SYSTEM Boiler
  (* Version 1.0, Author, 4DIAC-Consortium *)
  APPLICATION MyBoiler
    FBS
      IN_ANY_1 : IN_ANY(QI := 1, TYPE := LREAL, IVAL := 0);
      OUT_ANY : OUT_ANY(QI := 1, TYPE := LREAL, IVAL := 0);
      LREAL2LREAL_0 : LREAL2LREAL;
      FB_LABEL_0 : FB_LABEL(QI := 1, LABEL := Steam Removal (0..10));
      LREAL2LREAL_2 : LREAL2LREAL;
      OUT_ANY_0 : OUT_ANY(QI := 1, TYPE := LREAL, IVAL := 1);
      FB_LABEL_1 : FB_LABEL(QI := 1, LABEL := Actual Fill Level);
      FB_LABEL_2 : FB_LABEL(QI := 1, LABEL := Actual Feed Water Flow);
      OUT_ANY_1 : OUT_ANY(QI := 1, TYPE := LREAL, IVAL := 1);
      FB_LABEL_3 : FB_LABEL(QI := 1, LABEL := Actual Steam Flow);
      LREAL2LREAL_5 : LREAL2LREAL;
      IN_ANY : IN_ANY(QI := 1, TYPE := LREAL, IVAL := 0);
      FB_LABEL : FB_LABEL(QI := 1, LABEL := Set Fill Level (0..1000));
      LREAL2LREAL : LREAL2LREAL;
      LREAL2LREAL_1 : LREAL2LREAL;
      FlowController : FlowController;
      ControlComputation : ControlComputation;
      BasicAO : BasicAO(minEng := 0, maxEng := 10, minRaw := 0, maxRaw := 16#FFFF);
      FeedWaterValve : QW(QI := 1, PARAMS := %watervalve%);
      SteamValve : QW(QI := 1, PARAMS := %steamvalve%);
      BasicAO_0 : BasicAO(minEng := 0, maxEng := 10, minRaw := 0, maxRaw := 16#FFFF);
      LC : BasicPID(bReset := 0, fCtrlCycleTime := 0.01, fTv := 0, fTd := 0.01, fKp := 1, fTn := 0);
      BasicAI_1 : BasicAI(minEng := 0, maxEng := 1000, minRaw := 0, maxRaw := 16#FFFF);
      TankLevel : IW(QI := 1, PARAMS := %tanklevel%);
      E_CYCLE : E_CYCLE(DT := T#100ms);
      BasicAI_2 : BasicAI(minEng := 0, maxEng := 10, minRaw := 0, maxRaw := 16#FFFF);
      SteamFlow : IW(QI := 1, PARAMS := %steamflow%);
      IW : IW(QI := 1, PARAMS := %feedwaterflow%);
      BasicAI_3 : BasicAI(minEng := 0, maxEng := 10, minRaw := 0, maxRaw := 16#FFFF);
      LREAL2LREAL_3 : LREAL2LREAL;
      OUT_ANY_2 : OUT_ANY(QI := 1, TYPE := LREAL, IVAL := 0);
      FB_LABEL_4 : FB_LABEL(QI := 1, LABEL := Feed Water Valve);
      IN_ANY_0 : IN_ANY(TYPE := LREAL, IVAL := 0);
    END_FBS
    EVENT_CONNECTIONS
      LREAL2LREAL_0.CNF TO OUT_ANY.REQ;
      FB_LABEL_0.INITO TO IN_ANY_1.INIT;
      OUT_ANY.CNF TO LREAL2LREAL_2.REQ;
      LREAL2LREAL_2.CNF TO OUT_ANY_0.REQ;
      FB_LABEL_1.INITO TO OUT_ANY.INIT;
      OUT_ANY.INITO TO FB_LABEL_2.INIT;
      FB_LABEL_2.INITO TO OUT_ANY_0.INIT;
      FB_LABEL_3.INITO TO OUT_ANY_1.INIT;
      OUT_ANY_0.INITO TO FB_LABEL_3.INIT;
      LREAL2LREAL_5.CNF TO OUT_ANY_1.REQ;
      OUT_ANY_0.CNF TO LREAL2LREAL_5.REQ;
      FB_LABEL.INITO TO IN_ANY.INIT;
      IN_ANY.INITO TO FB_LABEL_0.INIT;
      IN_ANY.IND TO LREAL2LREAL.REQ;
      LREAL2LREAL.CNF TO IN_ANY_1.REQ;
      IN_ANY_1.IND TO LREAL2LREAL_1.REQ;
      ControlComputation.CNF TO FlowController.REQ;
      FlowController.CNF TO BasicAO.REQ;
      BasicAO.CNF TO FeedWaterValve.REQ;
      BasicAO.INITO TO FeedWaterValve.INIT;
      BasicAO_0.CNF TO SteamValve.REQ;
      BasicAO_0.INITO TO SteamValve.INIT;
      LREAL2LREAL_1.CNF TO BasicAO_0.REQ;
      TankLevel.INITO TO BasicAI_1.INIT;
      TankLevel.CNF TO BasicAI_1.REQ;
      E_CYCLE.EO TO TankLevel.REQ;
      LC.CNF TO ControlComputation.REQ;
      SteamFlow.CNF TO BasicAI_2.REQ;
      IW.CNF TO BasicAI_3.REQ;
      BasicAI_1.CNF TO IW.REQ;
      BasicAI_2.CNF TO LC.REQ;
      OUT_ANY_1.CNF TO LREAL2LREAL_3.REQ;
      LREAL2LREAL_3.CNF TO OUT_ANY_2.REQ;
      OUT_ANY_1.INITO TO FB_LABEL_4.INIT;
      FB_LABEL_4.INITO TO OUT_ANY_2.INIT;
      IW.INITO TO BasicAI_3.INIT;
      SteamFlow.INITO TO BasicAI_2.INIT;
      SteamValve.INITO TO BasicAO.INIT;
      BasicAI_3.CNF TO SteamFlow.REQ;
      BasicAI_3.INITO TO SteamFlow.INIT;
      BasicAI_1.INITO TO IW.INIT;
      BasicAI_2.INITO TO BasicAO_0.INIT;
      FeedWaterValve.INITO TO E_CYCLE.START;
    END_CONNECTIONS
    DATA_CONNECTIONS
      LREAL2LREAL_0.OUT TO OUT_ANY.IN;
      LREAL2LREAL_2.OUT TO OUT_ANY_0.IN;
      LREAL2LREAL_5.OUT TO OUT_ANY_1.IN;
      FB_LABEL_0.QO TO IN_ANY_1.QI;
      FB_LABEL.QO TO IN_ANY.QI;
      IN_ANY.OUT TO LREAL2LREAL.IN;
      IN_ANY_1.OUT TO LREAL2LREAL_1.IN;
      ControlComputation.ControlOut TO FlowController.Setpoint;
      BasicAO.Out TO FeedWaterValve.OUT;
      FlowController.ControlOut TO BasicAO.Val;
      BasicAO_0.Out TO SteamValve.OUT;
      LREAL2LREAL_1.OUT TO BasicAO_0.Val;
      LREAL2LREAL.OUT TO LC.fSetpointValue;
      TankLevel.IN TO BasicAI_1.Val;
      LC.fCtrlOutput TO ControlComputation.Input1;
      BasicAI_1.Out TO LC.fActualValue;
      SteamFlow.IN TO BasicAI_2.Val;
      IW.IN TO BasicAI_3.Val;
      BasicAI_2.Out TO ControlComputation.Input3;
      BasicAI_3.Out TO ControlComputation.Input2;
      LREAL2LREAL_3.OUT TO OUT_ANY_2.IN;
      FlowController.ControlOut TO LREAL2LREAL_3.IN;
      BasicAI_2.Out TO LREAL2LREAL_5.IN;
      BasicAI_1.Out TO LREAL2LREAL_0.IN;
      BasicAI_3.Out TO LREAL2LREAL_2.IN;
    END_CONNECTIONS
  END_APPLICATION
  APPLICATION globals
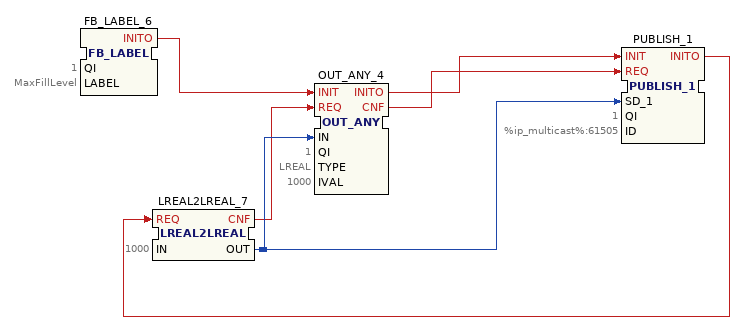
    FBS
      LREAL2LREAL_7 : LREAL2LREAL(IN := 1000);
      FB_LABEL_6 : FB_LABEL(QI := 1, LABEL := MaxFillLevel);
      OUT_ANY_4 : OUT_ANY(QI := 1, TYPE := LREAL, IVAL := 1000);
      PUBLISH_1 : PUBLISH_1(QI := 1, ID := %ip_multicast%:61505);
    END_FBS
    EVENT_CONNECTIONS
      OUT_ANY_4.INITO TO PUBLISH_1.INIT;
      FB_LABEL_6.INITO TO OUT_ANY_4.INIT;
      PUBLISH_1.INITO TO LREAL2LREAL_7.REQ;
      LREAL2LREAL_7.CNF TO OUT_ANY_4.REQ;
      OUT_ANY_4.CNF TO PUBLISH_1.REQ;
    END_CONNECTIONS
    DATA_CONNECTIONS
      LREAL2LREAL_7.OUT TO OUT_ANY_4.IN;
      LREAL2LREAL_7.OUT TO PUBLISH_1.SD_1;
    END_CONNECTIONS
  END_APPLICATION
  APPLICATION BoilerModel
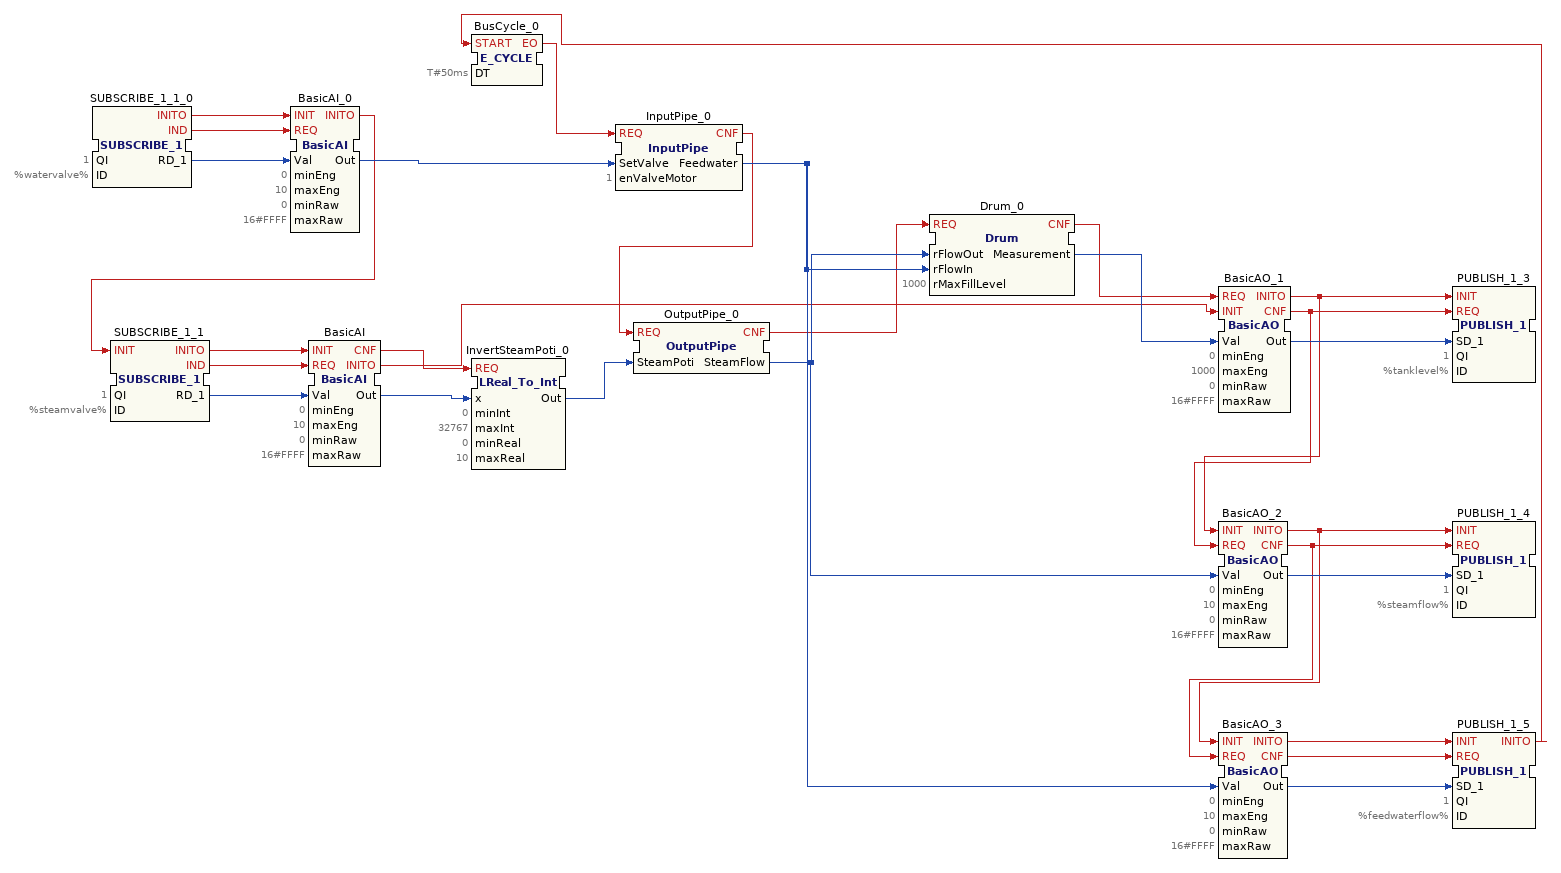
    FBS
      OutputPipe_0 : OutputPipe;
      Drum_0 : Drum(rMaxFillLevel := 1000);
      BusCycle_0 : E_CYCLE(DT := T#50ms);
      InvertSteamPoti_0 : LReal_To_Int(minInt := 0, maxInt := 32767, minReal := 0, maxReal := 10);
      InputPipe_0 : InputPipe(enValveMotor := 1);
      SUBSCRIBE_1_1 : SUBSCRIBE_1(QI := 1, ID := %steamvalve%);
      BasicAI : BasicAI(minEng := 0, maxEng := 10, minRaw := 0, maxRaw := 16#FFFF);
      SUBSCRIBE_1_1_0 : SUBSCRIBE_1(QI := 1, ID := %watervalve%);
      BasicAI_0 : BasicAI(minEng := 0, maxEng := 10, minRaw := 0, maxRaw := 16#FFFF);
      BasicAO_1 : BasicAO(minEng := 0, maxEng := 1000, minRaw := 0, maxRaw := 16#FFFF);
      BasicAO_2 : BasicAO(minEng := 0, maxEng := 10, minRaw := 0, maxRaw := 16#FFFF);
      BasicAO_3 : BasicAO(minEng := 0, maxEng := 10, minRaw := 0, maxRaw := 16#FFFF);
      PUBLISH_1_3 : PUBLISH_1(QI := 1, ID := %tanklevel%);
      PUBLISH_1_4 : PUBLISH_1(QI := 1, ID := %steamflow%);
      PUBLISH_1_5 : PUBLISH_1(QI := 1, ID := %feedwaterflow%);
    END_FBS
    EVENT_CONNECTIONS
      SUBSCRIBE_1_1.INITO TO BasicAI.INIT;
      SUBSCRIBE_1_1.IND TO BasicAI.REQ;
      SUBSCRIBE_1_1_0.INITO TO BasicAI_0.INIT;
      SUBSCRIBE_1_1_0.IND TO BasicAI_0.REQ;
      BasicAI.CNF TO InvertSteamPoti_0.REQ;
      BasicAO_1.INITO TO BasicAO_2.INIT;
      BasicAO_2.INITO TO BasicAO_3.INIT;
      BasicAO_1.CNF TO BasicAO_2.REQ;
      BasicAO_2.CNF TO BasicAO_3.REQ;
      BasicAO_1.INITO TO PUBLISH_1_3.INIT;
      BasicAO_1.CNF TO PUBLISH_1_3.REQ;
      BasicAO_2.INITO TO PUBLISH_1_4.INIT;
      BasicAO_2.CNF TO PUBLISH_1_4.REQ;
      BasicAO_3.INITO TO PUBLISH_1_5.INIT;
      BasicAO_3.CNF TO PUBLISH_1_5.REQ;
      BusCycle_0.EO TO InputPipe_0.REQ;
      OutputPipe_0.CNF TO Drum_0.REQ;
      InputPipe_0.CNF TO OutputPipe_0.REQ;
      BasicAI_0.INITO TO SUBSCRIBE_1_1.INIT;
      Drum_0.CNF TO BasicAO_1.REQ;
      PUBLISH_1_5.INITO TO BusCycle_0.START;
      BasicAI.INITO TO BasicAO_1.INIT;
    END_CONNECTIONS
    DATA_CONNECTIONS
      OutputPipe_0.SteamFlow TO Drum_0.rFlowOut;
      InputPipe_0.Feedwater TO Drum_0.rFlowIn;
      InvertSteamPoti_0.Out TO OutputPipe_0.SteamPoti;
      SUBSCRIBE_1_1.RD_1 TO BasicAI.Val;
      SUBSCRIBE_1_1_0.RD_1 TO BasicAI_0.Val;
      BasicAI_0.Out TO InputPipe_0.SetValve;
      BasicAI.Out TO InvertSteamPoti_0.x;
      BasicAO_1.Out TO PUBLISH_1_3.SD_1;
      BasicAO_2.Out TO PUBLISH_1_4.SD_1;
      BasicAO_3.Out TO PUBLISH_1_5.SD_1;
      Drum_0.Measurement TO BasicAO_1.Val;
      InputPipe_0.Feedwater TO BasicAO_3.Val;
      OutputPipe_0.SteamFlow TO BasicAO_2.Val;
    END_CONNECTIONS
  END_APPLICATION
  DEVICE HMI : FBRT_WINDOW(BOUNDS := [200,200,268,500], GRID := [3,1], MGR_ID := "localhost:61505")
    {SET_ATTRIBUTE(Profile, HOLOBLOC)}
    RESOURCE VIS_IN : PANEL_RESOURCE
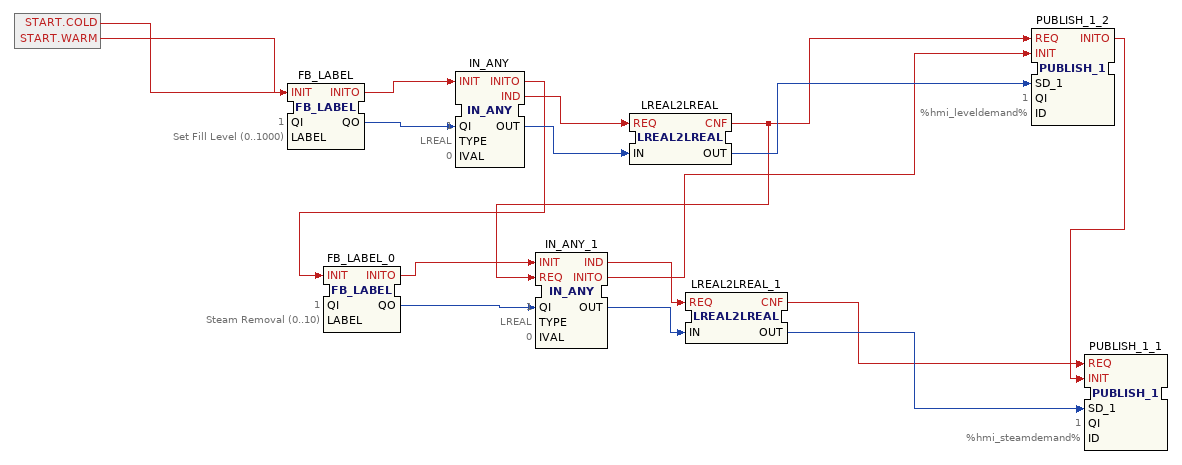
      FBS
        IN_ANY_1 : IN_ANY(QI := 1, TYPE := LREAL, IVAL := 0);
        FB_LABEL_0 : FB_LABEL(QI := 1, LABEL := Steam Removal (0..10));
        IN_ANY : IN_ANY(QI := 1, TYPE := LREAL, IVAL := 0);
        FB_LABEL : FB_LABEL(QI := 1, LABEL := Set Fill Level (0..1000));
        LREAL2LREAL : LREAL2LREAL;
        LREAL2LREAL_1 : LREAL2LREAL;
        PUBLISH_1_1 : PUBLISH_1(QI := 1, ID := %hmi_steamdemand%);
        PUBLISH_1_2 : PUBLISH_1(QI := 1, ID := %hmi_leveldemand%);
      END_FBS
      EVENT_CONNECTIONS
        FB_LABEL_0.INITO TO IN_ANY_1.INIT;
        IN_ANY.INITO TO FB_LABEL_0.INIT;
        FB_LABEL.INITO TO IN_ANY.INIT;
        IN_ANY.IND TO LREAL2LREAL.REQ;
        LREAL2LREAL.CNF TO IN_ANY_1.REQ;
        START.COLD TO FB_LABEL.INIT;
        START.WARM TO FB_LABEL.INIT;
        IN_ANY_1.IND TO LREAL2LREAL_1.REQ;
        LREAL2LREAL_1.CNF TO PUBLISH_1_1.REQ;
        LREAL2LREAL.CNF TO PUBLISH_1_2.REQ;
        IN_ANY_1.INITO TO PUBLISH_1_2.INIT;
        PUBLISH_1_2.INITO TO PUBLISH_1_1.INIT;
      END_CONNECTIONS
      DATA_CONNECTIONS
        FB_LABEL_0.QO TO IN_ANY_1.QI;
        FB_LABEL.QO TO IN_ANY.QI;
        IN_ANY.OUT TO LREAL2LREAL.IN;
        IN_ANY_1.OUT TO LREAL2LREAL_1.IN;
        LREAL2LREAL_1.OUT TO PUBLISH_1_1.SD_1;
        LREAL2LREAL.OUT TO PUBLISH_1_2.SD_1;
      END_CONNECTIONS
    END_RESOURCE
    RESOURCE VIS_OUT : PANEL_RESOURCE
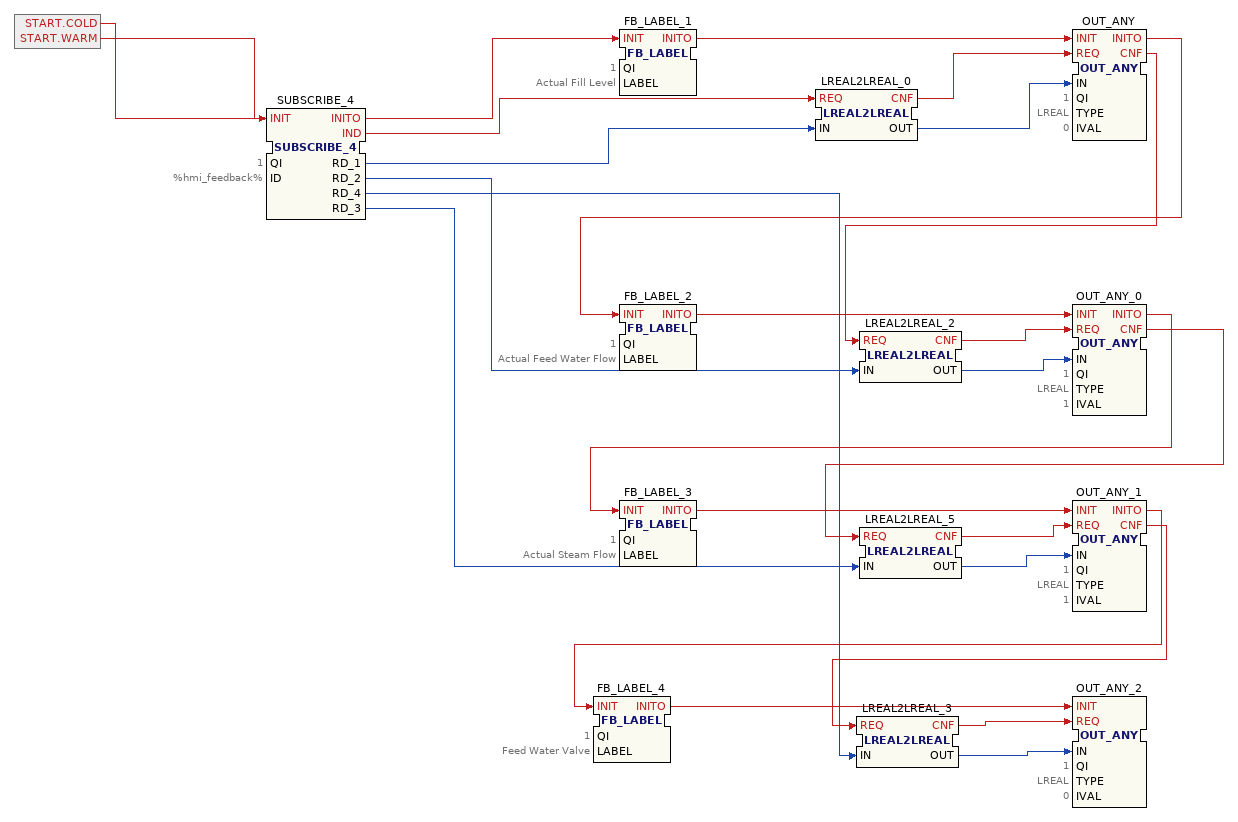
      FBS
        SUBSCRIBE_4 : SUBSCRIBE_4(QI := 1, ID := %hmi_feedback%);
        FB_LABEL_1 : FB_LABEL(QI := 1, LABEL := Actual Fill Level);
        LREAL2LREAL_0 : LREAL2LREAL;
        OUT_ANY : OUT_ANY(QI := 1, TYPE := LREAL, IVAL := 0);
        FB_LABEL_2 : FB_LABEL(QI := 1, LABEL := Actual Feed Water Flow);
        LREAL2LREAL_2 : LREAL2LREAL;
        OUT_ANY_0 : OUT_ANY(QI := 1, TYPE := LREAL, IVAL := 1);
        FB_LABEL_3 : FB_LABEL(QI := 1, LABEL := Actual Steam Flow);
        LREAL2LREAL_5 : LREAL2LREAL;
        OUT_ANY_1 : OUT_ANY(QI := 1, TYPE := LREAL, IVAL := 1);
        FB_LABEL_4 : FB_LABEL(QI := 1, LABEL := Feed Water Valve);
        LREAL2LREAL_3 : LREAL2LREAL;
        OUT_ANY_2 : OUT_ANY(QI := 1, TYPE := LREAL, IVAL := 0);
      END_FBS
      EVENT_CONNECTIONS
        START.COLD TO SUBSCRIBE_4.INIT;
        START.WARM TO SUBSCRIBE_4.INIT;
        FB_LABEL_1.INITO TO OUT_ANY.INIT;
        LREAL2LREAL_0.CNF TO OUT_ANY.REQ;
        OUT_ANY.INITO TO FB_LABEL_2.INIT;
        OUT_ANY.CNF TO LREAL2LREAL_2.REQ;
        FB_LABEL_2.INITO TO OUT_ANY_0.INIT;
        LREAL2LREAL_2.CNF TO OUT_ANY_0.REQ;
        OUT_ANY_0.INITO TO FB_LABEL_3.INIT;
        OUT_ANY_0.CNF TO LREAL2LREAL_5.REQ;
        FB_LABEL_3.INITO TO OUT_ANY_1.INIT;
        LREAL2LREAL_5.CNF TO OUT_ANY_1.REQ;
        OUT_ANY_1.INITO TO FB_LABEL_4.INIT;
        OUT_ANY_1.CNF TO LREAL2LREAL_3.REQ;
        FB_LABEL_4.INITO TO OUT_ANY_2.INIT;
        LREAL2LREAL_3.CNF TO OUT_ANY_2.REQ;
        SUBSCRIBE_4.INITO TO FB_LABEL_1.INIT;
        SUBSCRIBE_4.IND TO LREAL2LREAL_0.REQ;
      END_CONNECTIONS
      DATA_CONNECTIONS
        LREAL2LREAL_0.OUT TO OUT_ANY.IN;
        LREAL2LREAL_2.OUT TO OUT_ANY_0.IN;
        LREAL2LREAL_5.OUT TO OUT_ANY_1.IN;
        LREAL2LREAL_3.OUT TO OUT_ANY_2.IN;
        SUBSCRIBE_4.RD_1 TO LREAL2LREAL_0.IN;
        SUBSCRIBE_4.RD_2 TO LREAL2LREAL_2.IN;
        SUBSCRIBE_4.RD_4 TO LREAL2LREAL_3.IN;
        SUBSCRIBE_4.RD_3 TO LREAL2LREAL_5.IN;
      END_CONNECTIONS
    END_RESOURCE
    RESOURCE GLOBALS : PANEL_RESOURCE
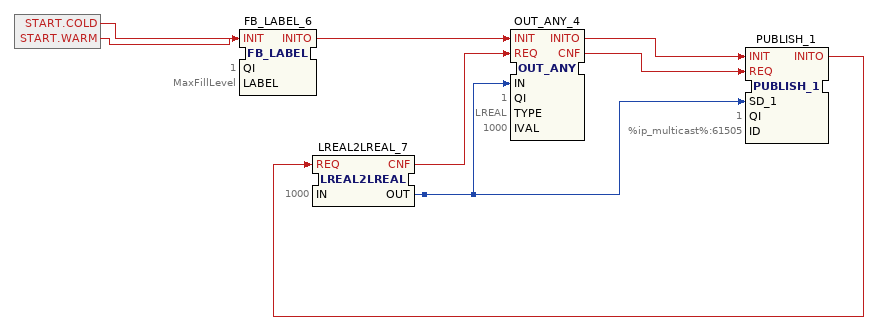
      FBS
        OUT_ANY_4 : OUT_ANY(QI := 1, TYPE := LREAL, IVAL := 1000);
        FB_LABEL_6 : FB_LABEL(QI := 1, LABEL := MaxFillLevel);
        LREAL2LREAL_7 : LREAL2LREAL(IN := 1000);
        PUBLISH_1 : PUBLISH_1(QI := 1, ID := %ip_multicast%:61505);
      END_FBS
      EVENT_CONNECTIONS
        START.COLD TO FB_LABEL_6.INIT;
        START.WARM TO FB_LABEL_6.INIT;
        OUT_ANY_4.INITO TO PUBLISH_1.INIT;
        FB_LABEL_6.INITO TO OUT_ANY_4.INIT;
        PUBLISH_1.INITO TO LREAL2LREAL_7.REQ;
        LREAL2LREAL_7.CNF TO OUT_ANY_4.REQ;
        OUT_ANY_4.CNF TO PUBLISH_1.REQ;
      END_CONNECTIONS
      DATA_CONNECTIONS
        LREAL2LREAL_7.OUT TO OUT_ANY_4.IN;
        LREAL2LREAL_7.OUT TO PUBLISH_1.SD_1;
      END_CONNECTIONS
    END_RESOURCE
  END_DEVICE
  DEVICE BoilerController : FORTE_PC(MGR_ID := %ip_controller%:61499)
    {SET_ATTRIBUTE(Profile, HOLOBLOC)}
    RESOURCE Controller : EMB_RES
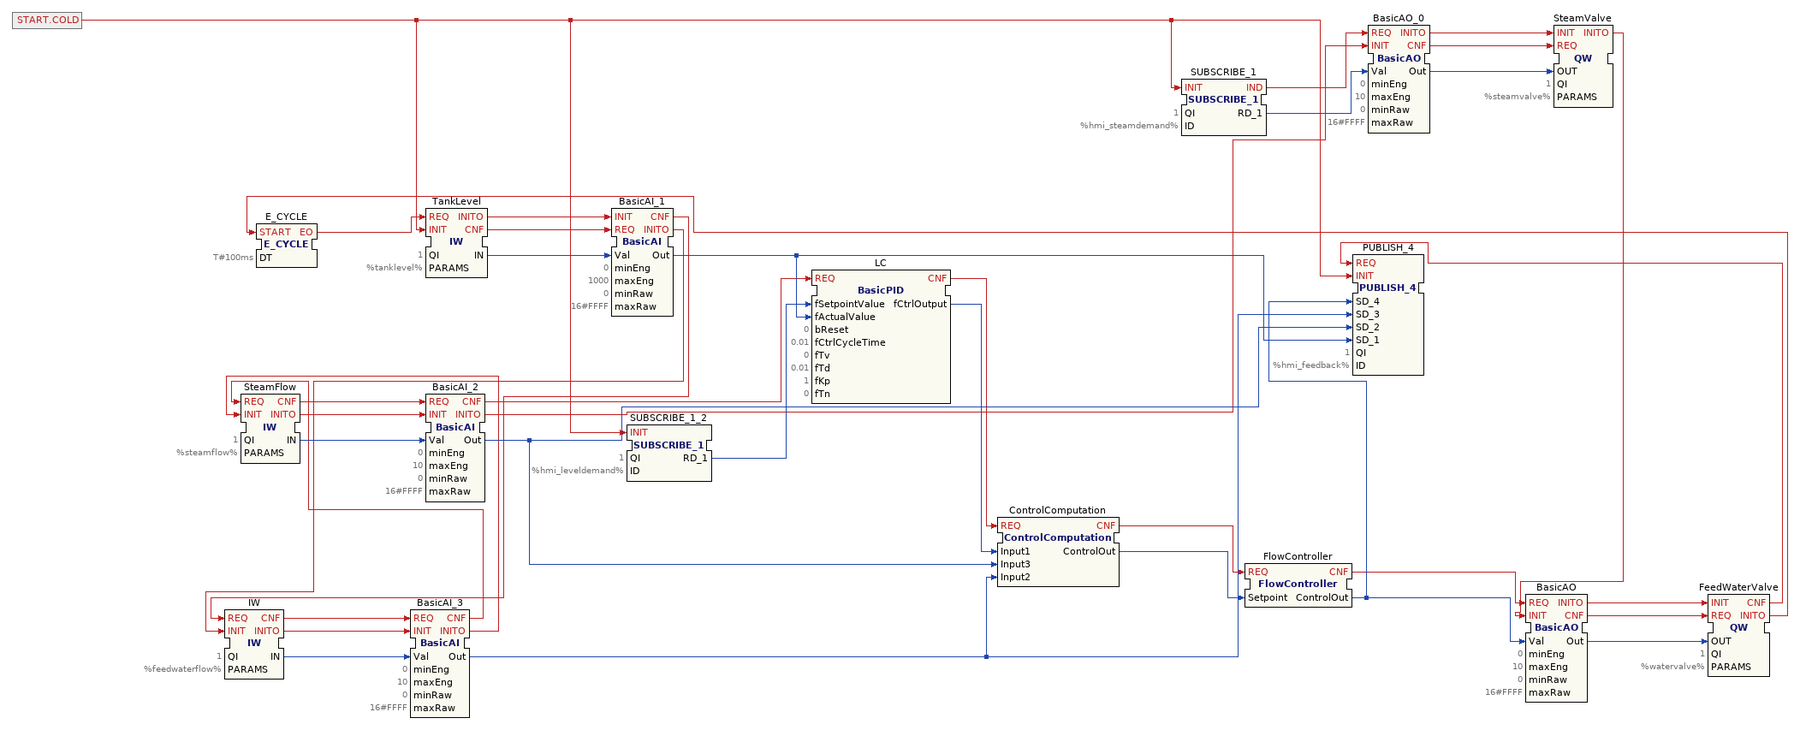
      FBS
        ControlComputation : ControlComputation;
        FlowController : FlowController;
        BasicAO : BasicAO(minEng := 0, maxEng := 10, minRaw := 0, maxRaw := 16#FFFF);
        FeedWaterValve : QW(QI := 1, PARAMS := %watervalve%);
        BasicAO_0 : BasicAO(minEng := 0, maxEng := 10, minRaw := 0, maxRaw := 16#FFFF);
        SteamValve : QW(QI := 1, PARAMS := %steamvalve%);
        SUBSCRIBE_1 : SUBSCRIBE_1(QI := 1, ID := %hmi_steamdemand%);
        TankLevel : IW(QI := 1, PARAMS := %tanklevel%);
        BasicAI_1 : BasicAI(minEng := 0, maxEng := 1000, minRaw := 0, maxRaw := 16#FFFF);
        LC : BasicPID(bReset := 0, fCtrlCycleTime := 0.01, fTv := 0, fTd := 0.01, fKp := 1, fTn := 0);
        E_CYCLE : E_CYCLE(DT := T#100ms);
        SUBSCRIBE_1_2 : SUBSCRIBE_1(QI := 1, ID := %hmi_leveldemand%);
        SteamFlow : IW(QI := 1, PARAMS := %steamflow%);
        BasicAI_2 : BasicAI(minEng := 0, maxEng := 10, minRaw := 0, maxRaw := 16#FFFF);
        IW : IW(QI := 1, PARAMS := %feedwaterflow%);
        BasicAI_3 : BasicAI(minEng := 0, maxEng := 10, minRaw := 0, maxRaw := 16#FFFF);
        PUBLISH_4 : PUBLISH_4(QI := 1, ID := %hmi_feedback%);
      END_FBS
      EVENT_CONNECTIONS
        ControlComputation.CNF TO FlowController.REQ;
        FlowController.CNF TO BasicAO.REQ;
        BasicAO.INITO TO FeedWaterValve.INIT;
        BasicAO.CNF TO FeedWaterValve.REQ;
        BasicAO_0.INITO TO SteamValve.INIT;
        BasicAO_0.CNF TO SteamValve.REQ;
        SUBSCRIBE_1.IND TO BasicAO_0.REQ;
        START.COLD TO SUBSCRIBE_1.INIT;
        TankLevel.INITO TO BasicAI_1.INIT;
        TankLevel.CNF TO BasicAI_1.REQ;
        E_CYCLE.EO TO TankLevel.REQ;
        LC.CNF TO ControlComputation.REQ;
        SteamFlow.CNF TO BasicAI_2.REQ;
        IW.CNF TO BasicAI_3.REQ;
        BasicAI_1.CNF TO IW.REQ;
        BasicAI_2.CNF TO LC.REQ;
        FeedWaterValve.CNF TO PUBLISH_4.REQ;
        IW.INITO TO BasicAI_3.INIT;
        SteamFlow.INITO TO BasicAI_2.INIT;
        SteamValve.INITO TO BasicAO.INIT;
        BasicAI_3.CNF TO SteamFlow.REQ;
        BasicAI_3.INITO TO SteamFlow.INIT;
        BasicAI_1.INITO TO IW.INIT;
        START.COLD TO TankLevel.INIT;
        START.COLD TO SUBSCRIBE_1_2.INIT;
        BasicAI_2.INITO TO BasicAO_0.INIT;
        FeedWaterValve.INITO TO E_CYCLE.START;
        START.COLD TO PUBLISH_4.INIT;
      END_CONNECTIONS
      DATA_CONNECTIONS
        ControlComputation.ControlOut TO FlowController.Setpoint;
        FlowController.ControlOut TO BasicAO.Val;
        BasicAO.Out TO FeedWaterValve.OUT;
        BasicAO_0.Out TO SteamValve.OUT;
        SUBSCRIBE_1.RD_1 TO BasicAO_0.Val;
        TankLevel.IN TO BasicAI_1.Val;
        SUBSCRIBE_1_2.RD_1 TO LC.fSetpointValue;
        LC.fCtrlOutput TO ControlComputation.Input1;
        BasicAI_1.Out TO LC.fActualValue;
        SteamFlow.IN TO BasicAI_2.Val;
        IW.IN TO BasicAI_3.Val;
        BasicAI_2.Out TO ControlComputation.Input3;
        BasicAI_3.Out TO ControlComputation.Input2;
        FlowController.ControlOut TO PUBLISH_4.SD_4;
        BasicAI_3.Out TO PUBLISH_4.SD_3;
        BasicAI_2.Out TO PUBLISH_4.SD_2;
        BasicAI_1.Out TO PUBLISH_4.SD_1;
      END_CONNECTIONS
    END_RESOURCE
  END_DEVICE
  DEVICE BoilerModel : FORTE_PC(MGR_ID := %ip_controller%:61498)
    {SET_ATTRIBUTE(Profile, HOLOBLOC)}
    RESOURCE Simulation : EMB_RES
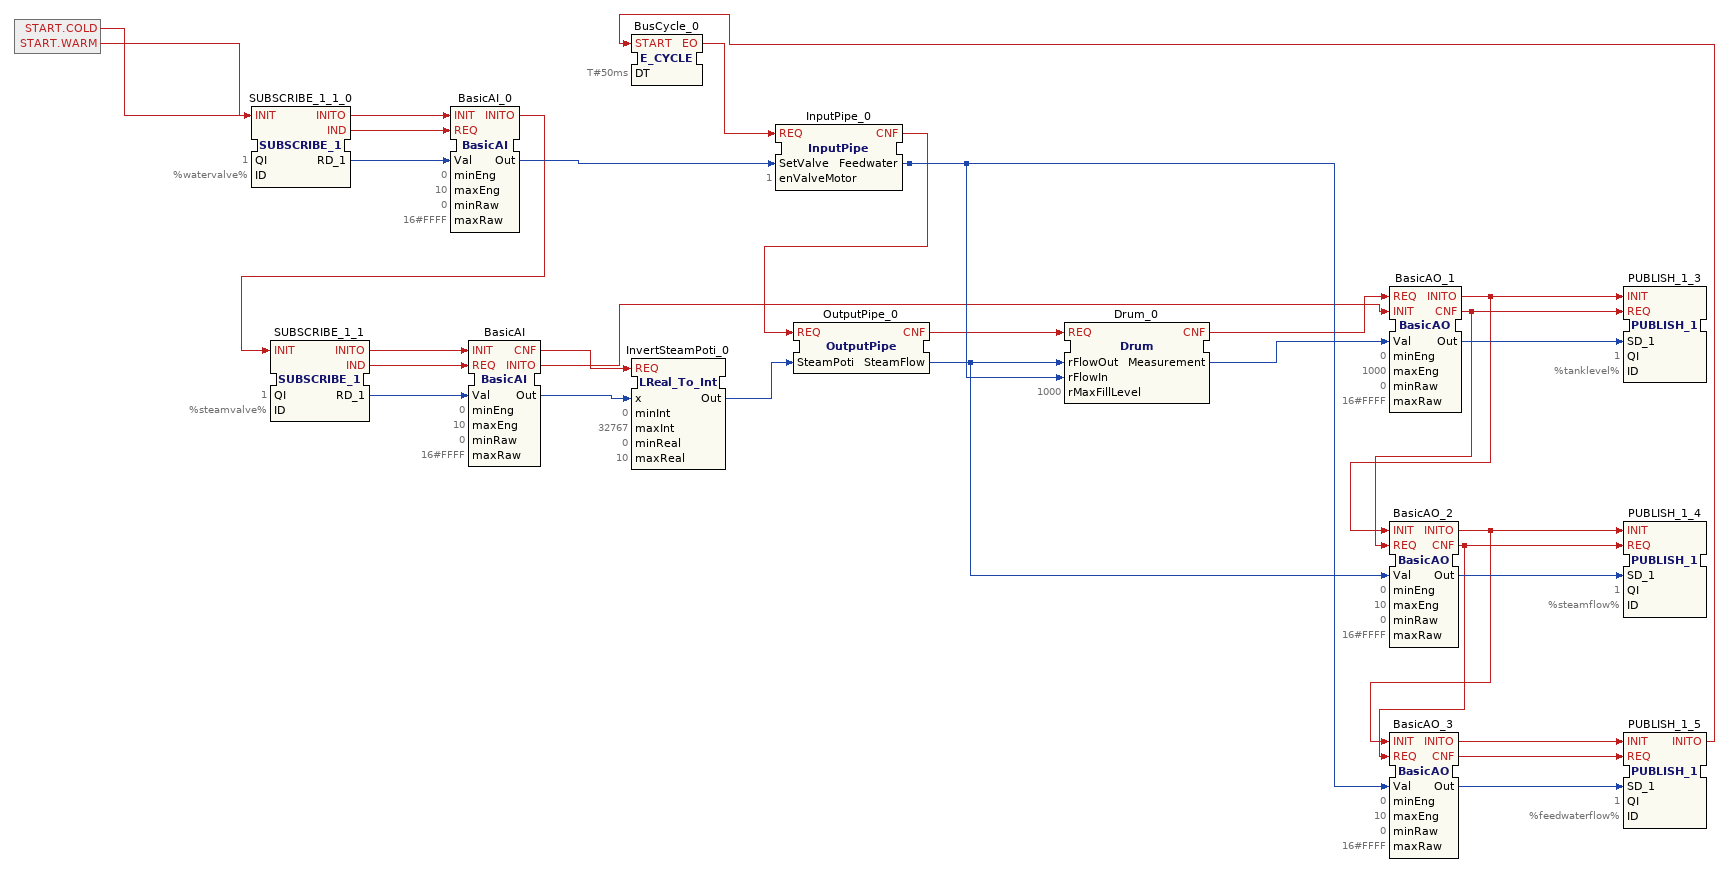
      FBS
        OutputPipe_0 : OutputPipe;
        Drum_0 : Drum(rMaxFillLevel := 1000);
        BusCycle_0 : E_CYCLE(DT := T#50ms);
        InvertSteamPoti_0 : LReal_To_Int(minInt := 0, maxInt := 32767, minReal := 0, maxReal := 10);
        InputPipe_0 : InputPipe(enValveMotor := 1);
        SUBSCRIBE_1_1 : SUBSCRIBE_1(QI := 1, ID := %steamvalve%);
        BasicAI : BasicAI(minEng := 0, maxEng := 10, minRaw := 0, maxRaw := 16#FFFF);
        SUBSCRIBE_1_1_0 : SUBSCRIBE_1(QI := 1, ID := %watervalve%);
        BasicAI_0 : BasicAI(minEng := 0, maxEng := 10, minRaw := 0, maxRaw := 16#FFFF);
        BasicAO_1 : BasicAO(minEng := 0, maxEng := 1000, minRaw := 0, maxRaw := 16#FFFF);
        BasicAO_2 : BasicAO(minEng := 0, maxEng := 10, minRaw := 0, maxRaw := 16#FFFF);
        BasicAO_3 : BasicAO(minEng := 0, maxEng := 10, minRaw := 0, maxRaw := 16#FFFF);
        PUBLISH_1_3 : PUBLISH_1(QI := 1, ID := %tanklevel%);
        PUBLISH_1_4 : PUBLISH_1(QI := 1, ID := %steamflow%);
        PUBLISH_1_5 : PUBLISH_1(QI := 1, ID := %feedwaterflow%);
      END_FBS
      EVENT_CONNECTIONS
        OutputPipe_0.CNF TO Drum_0.REQ;
        BusCycle_0.EO TO InputPipe_0.REQ;
        InputPipe_0.CNF TO OutputPipe_0.REQ;
        SUBSCRIBE_1_1.INITO TO BasicAI.INIT;
        SUBSCRIBE_1_1.IND TO BasicAI.REQ;
        BasicAI.CNF TO InvertSteamPoti_0.REQ;
        SUBSCRIBE_1_1_0.INITO TO BasicAI_0.INIT;
        SUBSCRIBE_1_1_0.IND TO BasicAI_0.REQ;
        BasicAI_0.INITO TO SUBSCRIBE_1_1.INIT;
        Drum_0.CNF TO BasicAO_1.REQ;
        BasicAO_1.INITO TO BasicAO_2.INIT;
        BasicAO_1.CNF TO BasicAO_2.REQ;
        BasicAO_2.INITO TO BasicAO_3.INIT;
        BasicAO_2.CNF TO BasicAO_3.REQ;
        BasicAO_1.INITO TO PUBLISH_1_3.INIT;
        BasicAO_1.CNF TO PUBLISH_1_3.REQ;
        BasicAO_2.INITO TO PUBLISH_1_4.INIT;
        BasicAO_2.CNF TO PUBLISH_1_4.REQ;
        BasicAO_3.INITO TO PUBLISH_1_5.INIT;
        BasicAO_3.CNF TO PUBLISH_1_5.REQ;
        START.COLD TO SUBSCRIBE_1_1_0.INIT;
        START.WARM TO SUBSCRIBE_1_1_0.INIT;
        PUBLISH_1_5.INITO TO BusCycle_0.START;
        BasicAI.INITO TO BasicAO_1.INIT;
      END_CONNECTIONS
      DATA_CONNECTIONS
        OutputPipe_0.SteamFlow TO Drum_0.rFlowOut;
        InvertSteamPoti_0.Out TO OutputPipe_0.SteamPoti;
        InputPipe_0.Feedwater TO Drum_0.rFlowIn;
        SUBSCRIBE_1_1.RD_1 TO BasicAI.Val;
        BasicAI.Out TO InvertSteamPoti_0.x;
        SUBSCRIBE_1_1_0.RD_1 TO BasicAI_0.Val;
        BasicAI_0.Out TO InputPipe_0.SetValve;
        Drum_0.Measurement TO BasicAO_1.Val;
        OutputPipe_0.SteamFlow TO BasicAO_2.Val;
        InputPipe_0.Feedwater TO BasicAO_3.Val;
        BasicAO_1.Out TO PUBLISH_1_3.SD_1;
        BasicAO_2.Out TO PUBLISH_1_4.SD_1;
        BasicAO_3.Out TO PUBLISH_1_5.SD_1;
      END_CONNECTIONS
    END_RESOURCE
  END_DEVICE
  MAPPINGS
    MyBoiler.IN_ANY_1 ON HMI.VIS_IN.IN_ANY_1;
    MyBoiler.OUT_ANY ON HMI.VIS_OUT.OUT_ANY;
    MyBoiler.LREAL2LREAL_0 ON HMI.VIS_OUT.LREAL2LREAL_0;
    MyBoiler.FB_LABEL_0 ON HMI.VIS_IN.FB_LABEL_0;
    MyBoiler.LREAL2LREAL_2 ON HMI.VIS_OUT.LREAL2LREAL_2;
    MyBoiler.OUT_ANY_0 ON HMI.VIS_OUT.OUT_ANY_0;
    MyBoiler.FB_LABEL_1 ON HMI.VIS_OUT.FB_LABEL_1;
    MyBoiler.FB_LABEL_2 ON HMI.VIS_OUT.FB_LABEL_2;
    MyBoiler.OUT_ANY_1 ON HMI.VIS_OUT.OUT_ANY_1;
    MyBoiler.FB_LABEL_3 ON HMI.VIS_OUT.FB_LABEL_3;
    MyBoiler.LREAL2LREAL_5 ON HMI.VIS_OUT.LREAL2LREAL_5;
    MyBoiler.IN_ANY ON HMI.VIS_IN.IN_ANY;
    MyBoiler.FB_LABEL ON HMI.VIS_IN.FB_LABEL;
    MyBoiler.LREAL2LREAL ON HMI.VIS_IN.LREAL2LREAL;
    MyBoiler.LREAL2LREAL_1 ON HMI.VIS_IN.LREAL2LREAL_1;
    MyBoiler.FlowController ON BoilerController.Controller.FlowController;
    MyBoiler.ControlComputation ON BoilerController.Controller.ControlComputation;
    MyBoiler.BasicAO ON BoilerController.Controller.BasicAO;
    MyBoiler.FeedWaterValve ON BoilerController.Controller.FeedWaterValve;
    MyBoiler.SteamValve ON BoilerController.Controller.SteamValve;
    MyBoiler.BasicAO_0 ON BoilerController.Controller.BasicAO_0;
    MyBoiler.LC ON BoilerController.Controller.LC;
    MyBoiler.BasicAI_1 ON BoilerController.Controller.BasicAI_1;
    MyBoiler.TankLevel ON BoilerController.Controller.TankLevel;
    MyBoiler.E_CYCLE ON BoilerController.Controller.E_CYCLE;
    MyBoiler.BasicAI_2 ON BoilerController.Controller.BasicAI_2;
    MyBoiler.SteamFlow ON BoilerController.Controller.SteamFlow;
    MyBoiler.IW ON BoilerController.Controller.IW;
    MyBoiler.BasicAI_3 ON BoilerController.Controller.BasicAI_3;
    MyBoiler.LREAL2LREAL_3 ON HMI.VIS_OUT.LREAL2LREAL_3;
    MyBoiler.OUT_ANY_2 ON HMI.VIS_OUT.OUT_ANY_2;
    MyBoiler.FB_LABEL_4 ON HMI.VIS_OUT.FB_LABEL_4;
    globals.LREAL2LREAL_7 ON HMI.GLOBALS.LREAL2LREAL_7;
    globals.FB_LABEL_6 ON HMI.GLOBALS.FB_LABEL_6;
    globals.OUT_ANY_4 ON HMI.GLOBALS.OUT_ANY_4;
    globals.PUBLISH_1 ON HMI.GLOBALS.PUBLISH_1;
    BoilerModel.OutputPipe_0 ON BoilerModel.Simulation.OutputPipe_0;
    BoilerModel.Drum_0 ON BoilerModel.Simulation.Drum_0;
    BoilerModel.BusCycle_0 ON BoilerModel.Simulation.BusCycle_0;
    BoilerModel.InvertSteamPoti_0 ON BoilerModel.Simulation.InvertSteamPoti_0;
    BoilerModel.InputPipe_0 ON BoilerModel.Simulation.InputPipe_0;
    BoilerModel.SUBSCRIBE_1_1 ON BoilerModel.Simulation.SUBSCRIBE_1_1;
    BoilerModel.BasicAI ON BoilerModel.Simulation.BasicAI;
    BoilerModel.SUBSCRIBE_1_1_0 ON BoilerModel.Simulation.SUBSCRIBE_1_1_0;
    BoilerModel.BasicAI_0 ON BoilerModel.Simulation.BasicAI_0;
    BoilerModel.BasicAO_1 ON BoilerModel.Simulation.BasicAO_1;
    BoilerModel.BasicAO_2 ON BoilerModel.Simulation.BasicAO_2;
    BoilerModel.BasicAO_3 ON BoilerModel.Simulation.BasicAO_3;
    BoilerModel.PUBLISH_1_3 ON BoilerModel.Simulation.PUBLISH_1_3;
    BoilerModel.PUBLISH_1_4 ON BoilerModel.Simulation.PUBLISH_1_4;
    BoilerModel.PUBLISH_1_5 ON BoilerModel.Simulation.PUBLISH_1_5;
  END_MAPPINGS
  SEGMENTS
    Ethernet : Ethernet;
  END_SEGMENTS
  LINKS
    HMI => Ethernet;
    BoilerController => Ethernet;
    BoilerModel => Ethernet;
  END_LINKS
END_SYSTEM
